(* Logix 5000 project; controller cal1615 1756-L62 rev 20.19; software revision 20.05; part 35 of 81 *)
(* tags used below, declared in another part *)
   FAULT : BOOL;   // Fault AFI
   HMI : BOOL;   // AFI HMI
   p01_param_oven_timer_presets : DINT[32];   // System Parameter Oven Timer Presets
   p01_sys_lc : Limit_Clamp;   // Zone 1 Misc Control Limit Clamp
   p01r09_pb_global_reset : BOOL;   // System Modes PB: Global Fault Reset
   p01r11 : routine;   // System Timer Presets
   p02_real_from_hmi : hmi_real;   // MOP HMI Iface Real from HMI
   p19_dint_to_hmi : DINT[16];
   p19_param_pid1_ff : REAL;
   p19_param_pid1_kd : REAL;
   p19_param_pid1_ki : REAL;
   p19_param_pid1_kp : REAL;
   p19_param_pid2_ff : REAL;
   p19_param_pid2_kd : REAL;
   p19_param_pid2_ki : REAL;
   p19_param_pid2_kp : REAL;
   p19_param_tc01_dev : REAL;
   p19_param_tc01z : REAL;   // Advanced Cooling Parameter Control Temperature 1 Zero Offset
   p19_param_tc02z : REAL;   // Advanced Cooling Parameter Control Temperature 2 Zero Offset
   p19_param_zone_pressure : REAL;   // Advanced Cooling Parameter Minimum Pressusre
   p19r01 : routine;   // Advanced Cooling Main
   p19r02_timer_warning : TIMER[4];   // Advanced Cooling Warning Delay
   p19r07 : routine;   // Advanced Cooling Alarms
   p19r07_timer_fault : TIMER[4];   // Advanced Cooling Alarms Fault Delay
   p19r07_timer_warning : TIMER[4];   // Advanced Cooling Alarms Warning Delay
   p19r08 : routine;   // Advanced Cooling Warnings
   p19r08_timer_fault : TIMER[4];   // Advanced Cooling Warnings Fault Delay
   p19r08_timer_warning : TIMER[4];   // Advanced Cooling Warnings Warning Delay
   p19r09 : routine;   // Advanced Cooling Modes
   p19r09_timer_fault : TIMER[4];   // Advanced Cooling Modes Fault Delay
   p19r09_timer_warning : TIMER[4];   // Advanced Cooling Modes Warning Delay
   p19r10 : routine;   // Advanced Cooling Parameters
   p19r10_timer_fault : TIMER[4];   // Advanced Cooling Parameters Fault Delay
   p19r30 : routine;   // Advanced Cooling Temperature Control
   p19r30_cv_man_sp : REAL;   // Advanced Cooling Manual Control Valve Setpoint
   p19r30_timer_fault : TIMER[4];   // Advanced Cooling Temperature Control Thermocouple Failure
   p19r30_timer_warning : TIMER[4];   // Advanced Cooling Temperature Control Warning Delay
   p19r31 : routine;   // Advanced Cooling Pump
   p19r31_timer_fault : TIMER[4];   // Advanced Cooling Pump Fault Delay
(* P19_Advanced_Cooling, continued *)

ROUTINE R07_Alarms   (* ladder *)
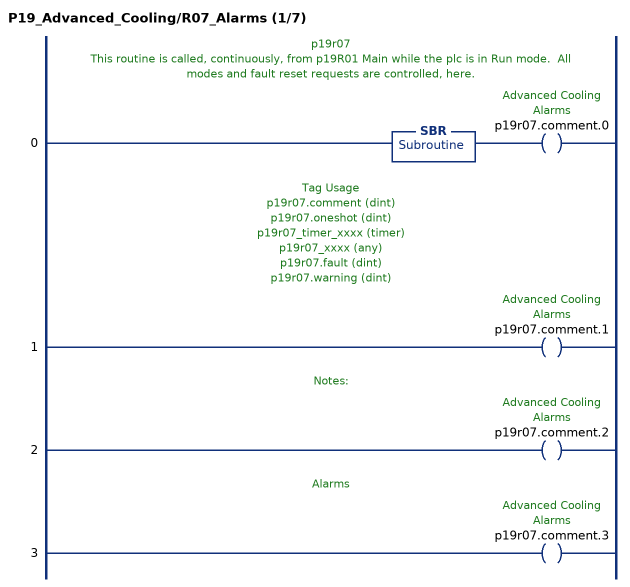
   // p19r07
   // This routine is called, continuously, from p19R01 Main while the plc is in Run mode.  All modes and fault reset requests are controlled, here.
   0: SBR()OTE(p19r07.comment.0);
   // Tag Usage
   // p19r07.comment (dint)
   // p19r07.oneshot (dint)
   // p19r07_timer_xxxx (timer)
   // p19r07_xxxx (any)
   // p19r07.fault (dint)
   // p19r07.warning (dint)
   1: OTE(p19r07.comment.1);
   // Notes:
   2: OTE(p19r07.comment.2);
   // Alarms
   3: OTE(p19r07.comment.3);
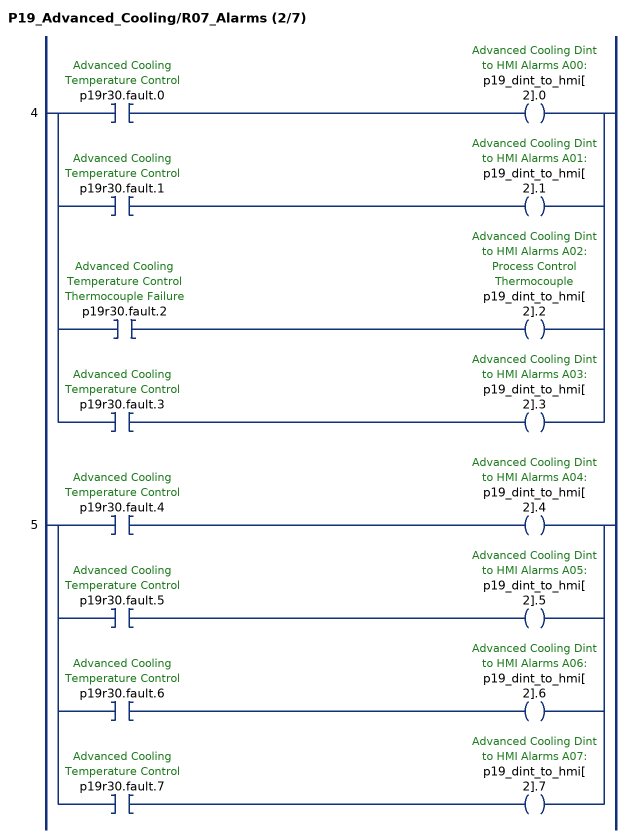
   4: [XIC(p19r30.fault.0) OTE(p19_dint_to_hmi[2].0) ,XIC(p19r30.fault.1) OTE(p19_dint_to_hmi[2].1) ,XIC(p19r30.fault.2) OTE(p19_dint_to_hmi[2].2) ,XIC(p19r30.fault.3) OTE(p19_dint_to_hmi[2].3) ];
   5: [XIC(p19r30.fault.4) OTE(p19_dint_to_hmi[2].4) ,XIC(p19r30.fault.5) OTE(p19_dint_to_hmi[2].5) ,XIC(p19r30.fault.6) OTE(p19_dint_to_hmi[2].6) ,XIC(p19r30.fault.7) OTE(p19_dint_to_hmi[2].7) ];
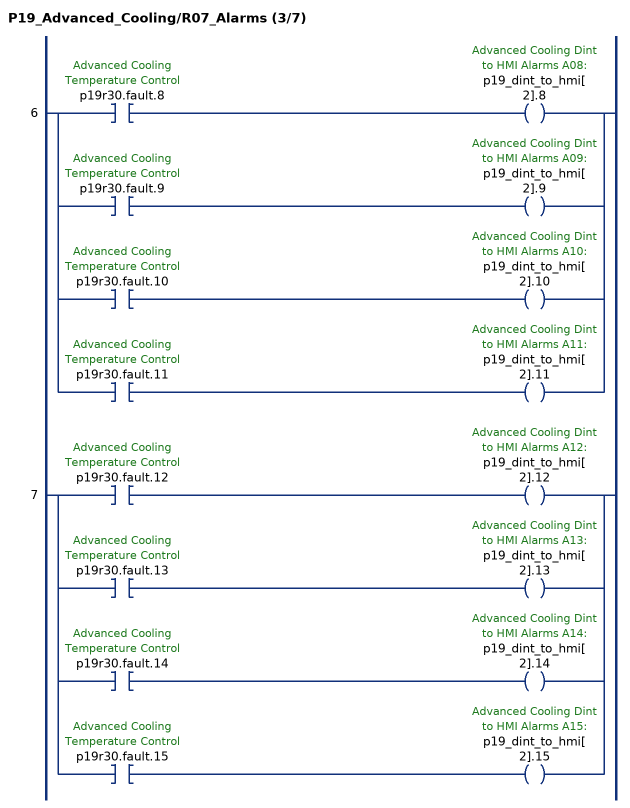
   6: [XIC(p19r30.fault.8) OTE(p19_dint_to_hmi[2].8) ,XIC(p19r30.fault.9) OTE(p19_dint_to_hmi[2].9) ,XIC(p19r30.fault.10) OTE(p19_dint_to_hmi[2].10) ,XIC(p19r30.fault.11) OTE(p19_dint_to_hmi[2].11) ];
   7: [XIC(p19r30.fault.12) OTE(p19_dint_to_hmi[2].12) ,XIC(p19r30.fault.13) OTE(p19_dint_to_hmi[2].13) ,XIC(p19r30.fault.14) OTE(p19_dint_to_hmi[2].14) ,XIC(p19r30.fault.15) OTE(p19_dint_to_hmi[2].15) ];
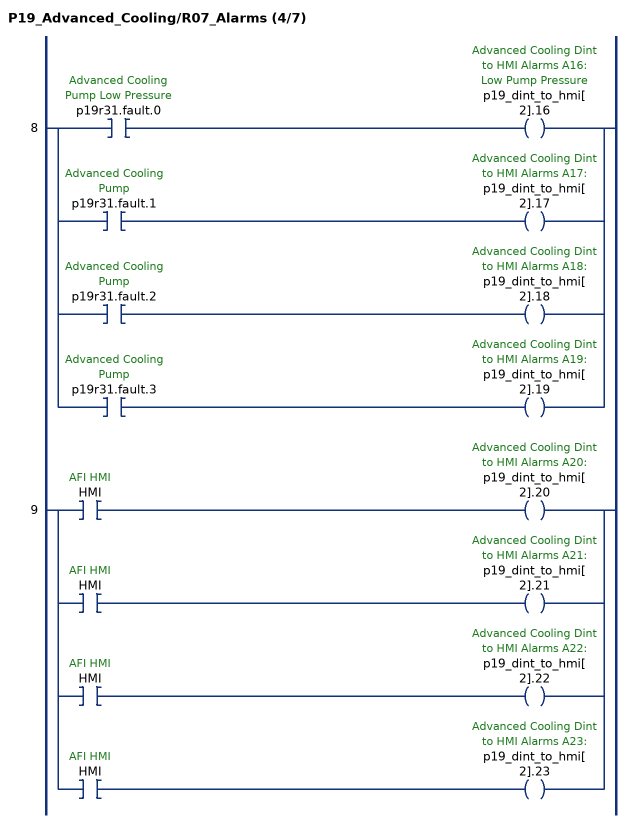
   8: [XIC(p19r31.fault.0) OTE(p19_dint_to_hmi[2].16) ,XIC(p19r31.fault.1) OTE(p19_dint_to_hmi[2].17) ,XIC(p19r31.fault.2) OTE(p19_dint_to_hmi[2].18) ,XIC(p19r31.fault.3) OTE(p19_dint_to_hmi[2].19) ];
   9: [XIC(HMI) OTE(p19_dint_to_hmi[2].20) ,XIC(HMI) OTE(p19_dint_to_hmi[2].21) ,XIC(HMI) OTE(p19_dint_to_hmi[2].22) ,XIC(HMI) OTE(p19_dint_to_hmi[2].23) ];
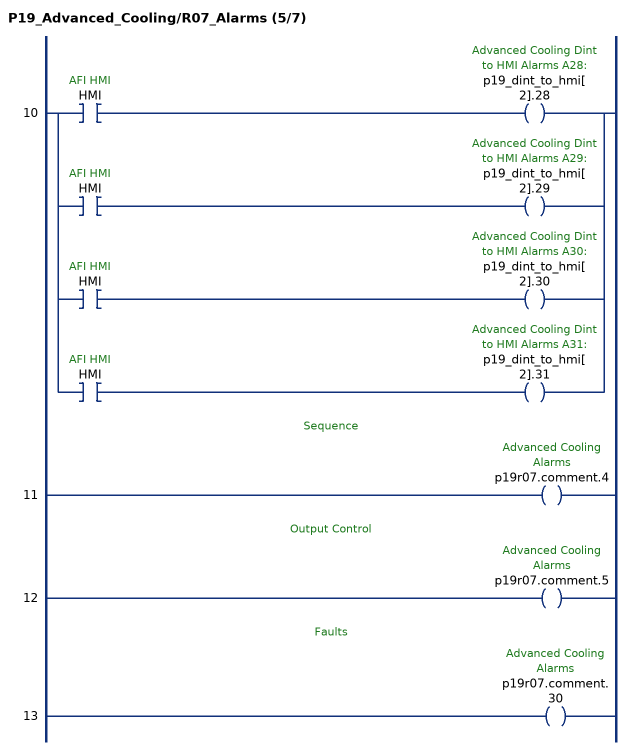
   10: [XIC(HMI) OTE(p19_dint_to_hmi[2].28) ,XIC(HMI) OTE(p19_dint_to_hmi[2].29) ,XIC(HMI) OTE(p19_dint_to_hmi[2].30) ,XIC(HMI) OTE(p19_dint_to_hmi[2].31) ];
   // Sequence
   11: OTE(p19r07.comment.4);
   // Output Control
   12: OTE(p19r07.comment.5);
   // Faults
   13: OTE(p19r07.comment.30);
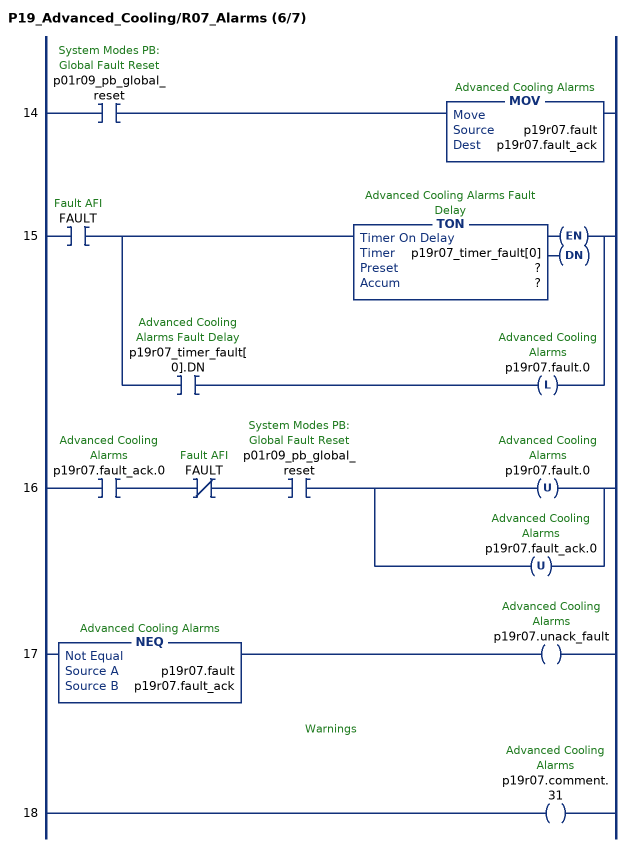
   14: XIC(p01r09_pb_global_reset)MOV(p19r07.fault,p19r07.fault_ack);
   15: XIC(FAULT)[TON(p19r07_timer_fault[0],?,?) ,XIC(p19r07_timer_fault[0].DN) OTL(p19r07.fault.0) ];
   16: XIC(p19r07.fault_ack.0)XIO(FAULT)XIC(p01r09_pb_global_reset)[OTU(p19r07.fault.0) ,OTU(p19r07.fault_ack.0) ];
   17: NEQ(p19r07.fault,p19r07.fault_ack)OTE(p19r07.unack_fault);
   // Warnings
   18: OTE(p19r07.comment.31);
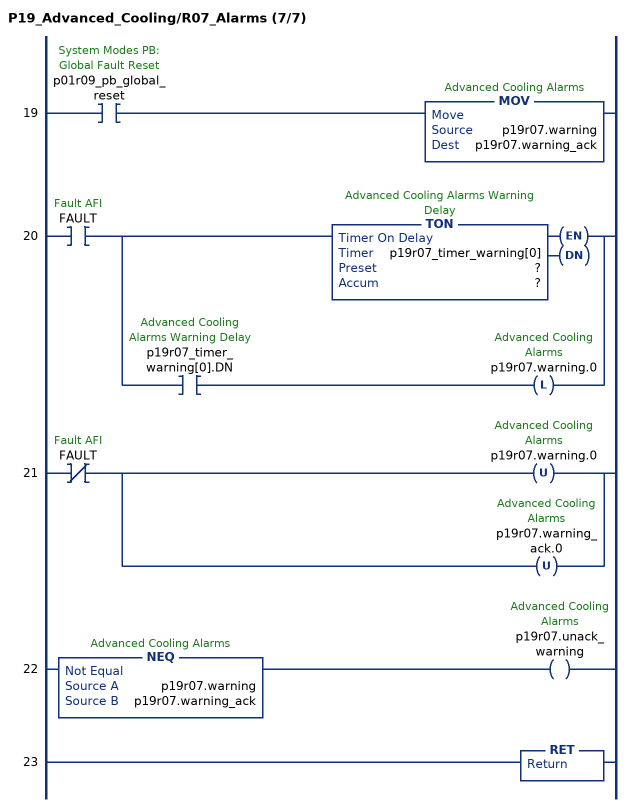
   19: XIC(p01r09_pb_global_reset)MOV(p19r07.warning,p19r07.warning_ack);
   20: XIC(FAULT)[TON(p19r07_timer_warning[0],?,?) ,XIC(p19r07_timer_warning[0].DN) OTL(p19r07.warning.0) ];
   21: XIO(FAULT)[OTU(p19r07.warning.0) ,OTU(p19r07.warning_ack.0) ];
   22: NEQ(p19r07.warning,p19r07.warning_ack)OTE(p19r07.unack_warning);
   23: RET();
END_ROUTINE

ROUTINE R08_Warnings   (* ladder *)
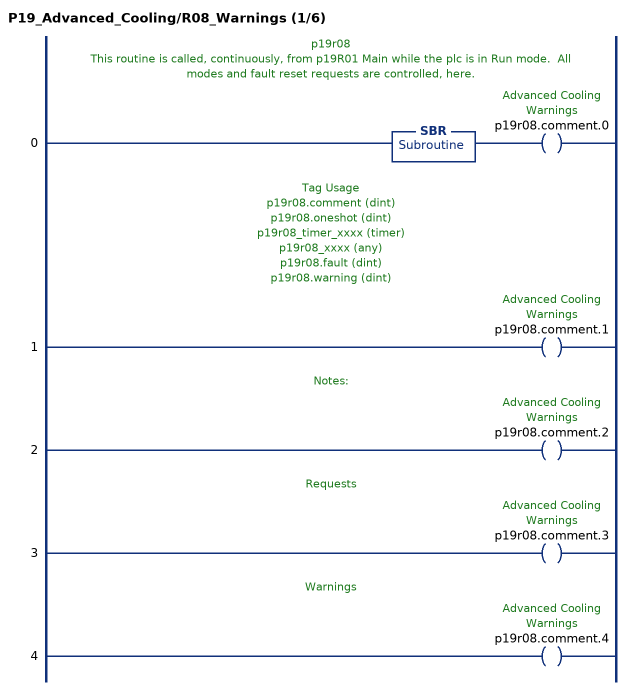
   // p19r08
   // This routine is called, continuously, from p19R01 Main while the plc is in Run mode.  All modes and fault reset requests are controlled, here.
   0: SBR()OTE(p19r08.comment.0);
   // Tag Usage
   // p19r08.comment (dint)
   // p19r08.oneshot (dint)
   // p19r08_timer_xxxx (timer)
   // p19r08_xxxx (any)
   // p19r08.fault (dint)
   // p19r08.warning (dint)
   1: OTE(p19r08.comment.1);
   // Notes:
   2: OTE(p19r08.comment.2);
   // Requests
   3: OTE(p19r08.comment.3);
   // Warnings
   4: OTE(p19r08.comment.4);
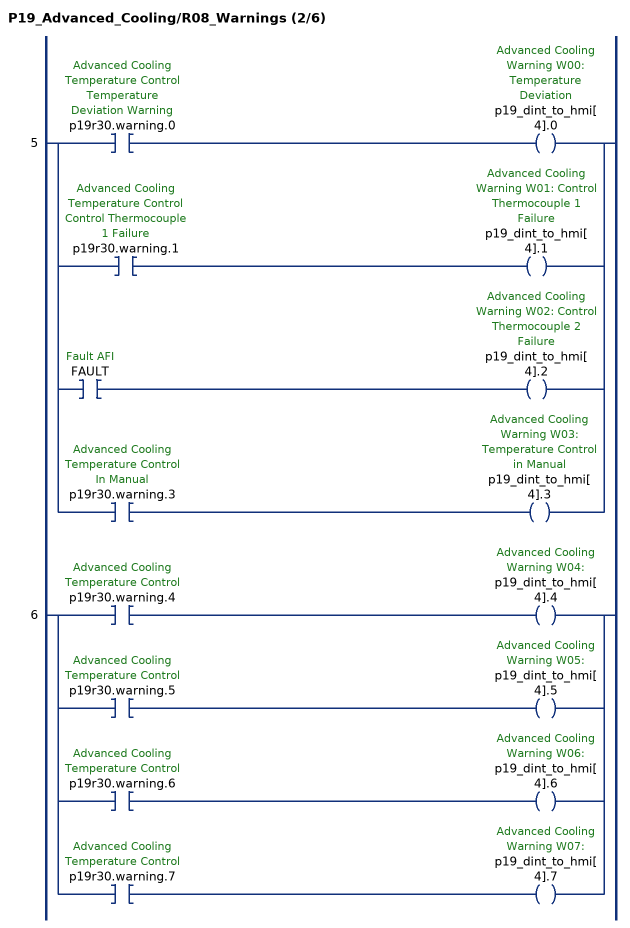
   5: [XIC(p19r30.warning.0) OTE(p19_dint_to_hmi[4].0) ,XIC(p19r30.warning.1) OTE(p19_dint_to_hmi[4].1) ,XIC(FAULT) OTE(p19_dint_to_hmi[4].2) ,XIC(p19r30.warning.3) OTE(p19_dint_to_hmi[4].3) ];
   6: [XIC(p19r30.warning.4) OTE(p19_dint_to_hmi[4].4) ,XIC(p19r30.warning.5) OTE(p19_dint_to_hmi[4].5) ,XIC(p19r30.warning.6) OTE(p19_dint_to_hmi[4].6) ,XIC(p19r30.warning.7) OTE(p19_dint_to_hmi[4].7) ];
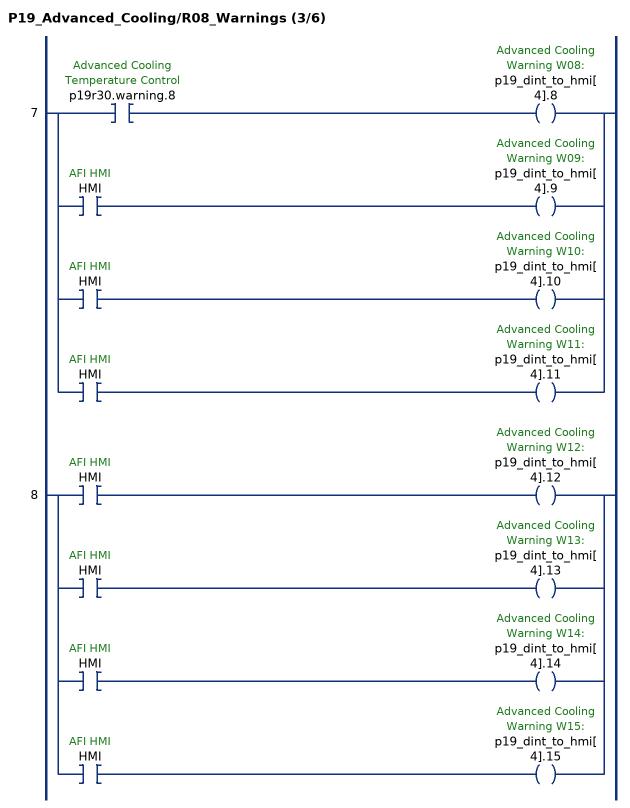
   7: [XIC(p19r30.warning.8) OTE(p19_dint_to_hmi[4].8) ,XIC(HMI) OTE(p19_dint_to_hmi[4].9) ,XIC(HMI) OTE(p19_dint_to_hmi[4].10) ,XIC(HMI) OTE(p19_dint_to_hmi[4].11) ];
   8: [XIC(HMI) OTE(p19_dint_to_hmi[4].12) ,XIC(HMI) OTE(p19_dint_to_hmi[4].13) ,XIC(HMI) OTE(p19_dint_to_hmi[4].14) ,XIC(HMI) OTE(p19_dint_to_hmi[4].15) ];
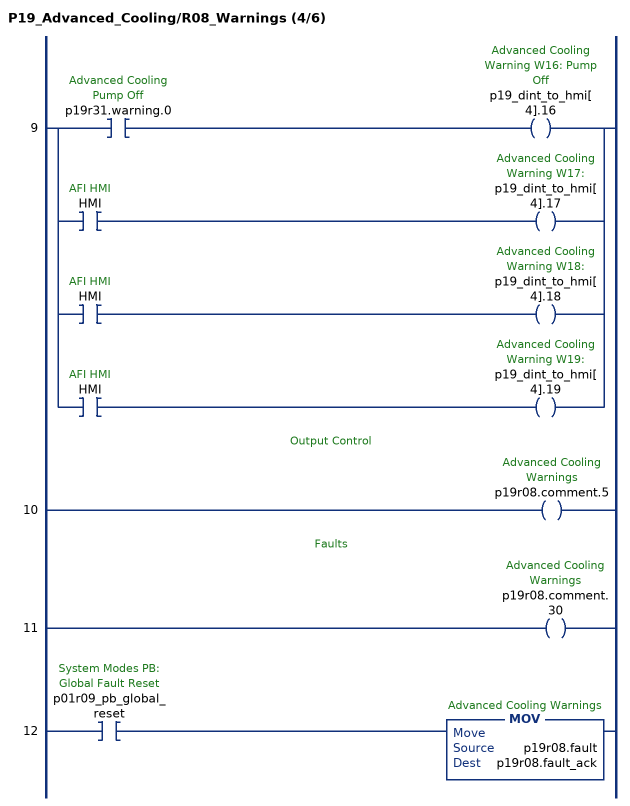
   9: [XIC(p19r31.warning.0) OTE(p19_dint_to_hmi[4].16) ,XIC(HMI) OTE(p19_dint_to_hmi[4].17) ,XIC(HMI) OTE(p19_dint_to_hmi[4].18) ,XIC(HMI) OTE(p19_dint_to_hmi[4].19) ];
   // Output Control
   10: OTE(p19r08.comment.5);
   // Faults
   11: OTE(p19r08.comment.30);
   12: XIC(p01r09_pb_global_reset)MOV(p19r08.fault,p19r08.fault_ack);
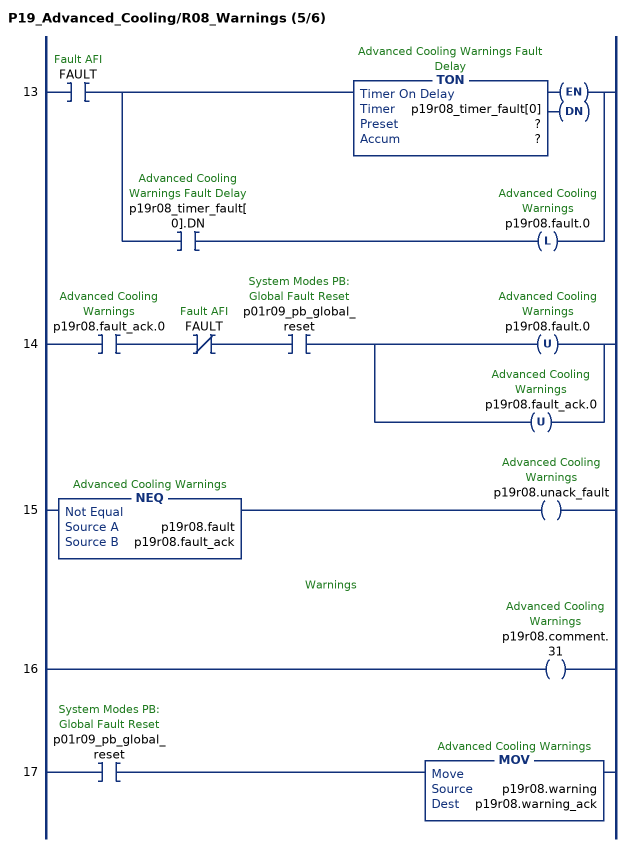
   13: XIC(FAULT)[TON(p19r08_timer_fault[0],?,?) ,XIC(p19r08_timer_fault[0].DN) OTL(p19r08.fault.0) ];
   14: XIC(p19r08.fault_ack.0)XIO(FAULT)XIC(p01r09_pb_global_reset)[OTU(p19r08.fault.0) ,OTU(p19r08.fault_ack.0) ];
   15: NEQ(p19r08.fault,p19r08.fault_ack)OTE(p19r08.unack_fault);
   // Warnings
   16: OTE(p19r08.comment.31);
   17: XIC(p01r09_pb_global_reset)MOV(p19r08.warning,p19r08.warning_ack);
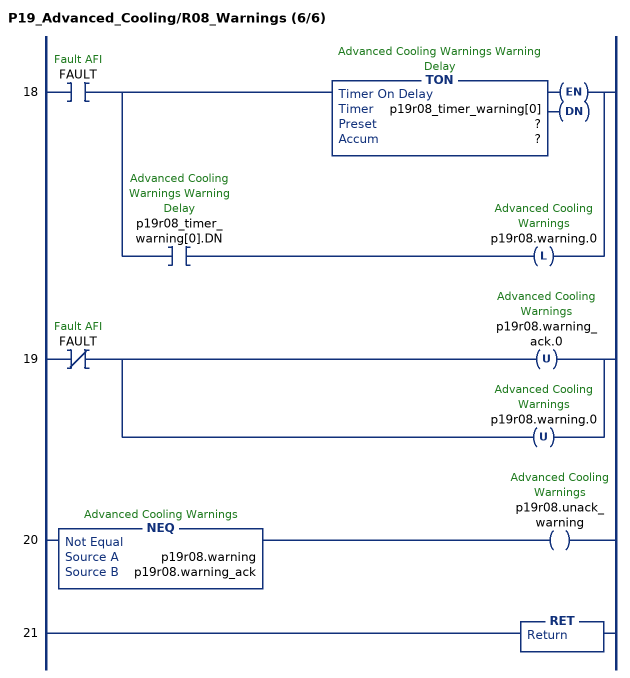
   18: XIC(FAULT)[TON(p19r08_timer_warning[0],?,?) ,XIC(p19r08_timer_warning[0].DN) OTL(p19r08.warning.0) ];
   19: XIO(FAULT)[OTU(p19r08.warning_ack.0) ,OTU(p19r08.warning.0) ];
   20: NEQ(p19r08.warning,p19r08.warning_ack)OTE(p19r08.unack_warning);
   21: RET();
END_ROUTINE

ROUTINE R09_Modes   (* ladder *)
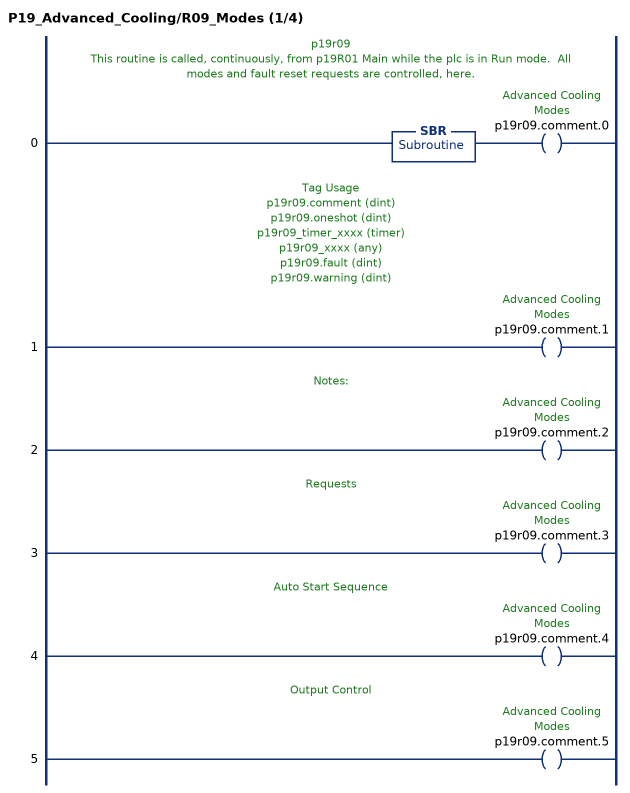
   // p19r09
   // This routine is called, continuously, from p19R01 Main while the plc is in Run mode.  All modes and fault reset requests are controlled, here.
   0: SBR()OTE(p19r09.comment.0);
   // Tag Usage
   // p19r09.comment (dint)
   // p19r09.oneshot (dint)
   // p19r09_timer_xxxx (timer)
   // p19r09_xxxx (any)
   // p19r09.fault (dint)
   // p19r09.warning (dint)
   1: OTE(p19r09.comment.1);
   // Notes:
   2: OTE(p19r09.comment.2);
   // Requests
   3: OTE(p19r09.comment.3);
   // Auto Start Sequence
   4: OTE(p19r09.comment.4);
   // Output Control
   5: OTE(p19r09.comment.5);
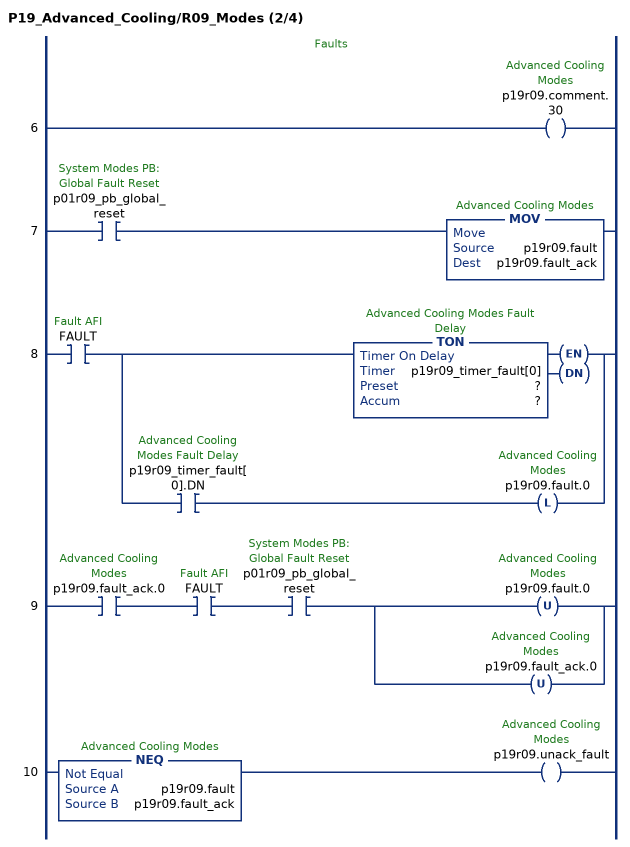
   // Faults
   6: OTE(p19r09.comment.30);
   7: XIC(p01r09_pb_global_reset)MOV(p19r09.fault,p19r09.fault_ack);
   8: XIC(FAULT)[TON(p19r09_timer_fault[0],?,?) ,XIC(p19r09_timer_fault[0].DN) OTL(p19r09.fault.0) ];
   9: XIC(p19r09.fault_ack.0)XIC(FAULT)XIC(p01r09_pb_global_reset)[OTU(p19r09.fault.0) ,OTU(p19r09.fault_ack.0) ];
   10: NEQ(p19r09.fault,p19r09.fault_ack)OTE(p19r09.unack_fault);
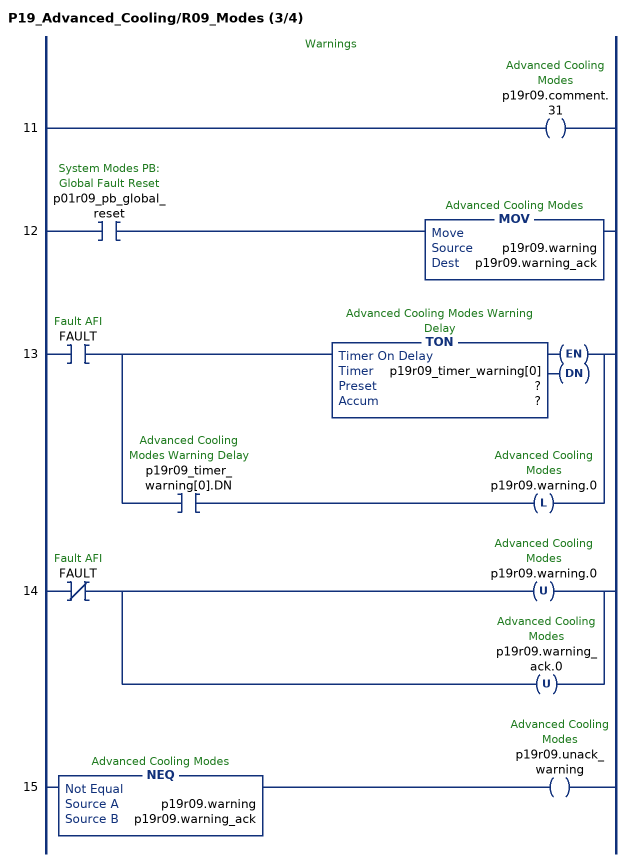
   // Warnings
   11: OTE(p19r09.comment.31);
   12: XIC(p01r09_pb_global_reset)MOV(p19r09.warning,p19r09.warning_ack);
   13: XIC(FAULT)[TON(p19r09_timer_warning[0],?,?) ,XIC(p19r09_timer_warning[0].DN) OTL(p19r09.warning.0) ];
   14: XIO(FAULT)[OTU(p19r09.warning.0) ,OTU(p19r09.warning_ack.0) ];
   15: NEQ(p19r09.warning,p19r09.warning_ack)OTE(p19r09.unack_warning);
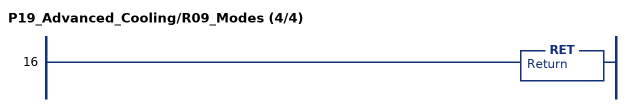
   16: RET();
END_ROUTINE

ROUTINE R10_Parameters   (* ladder *)
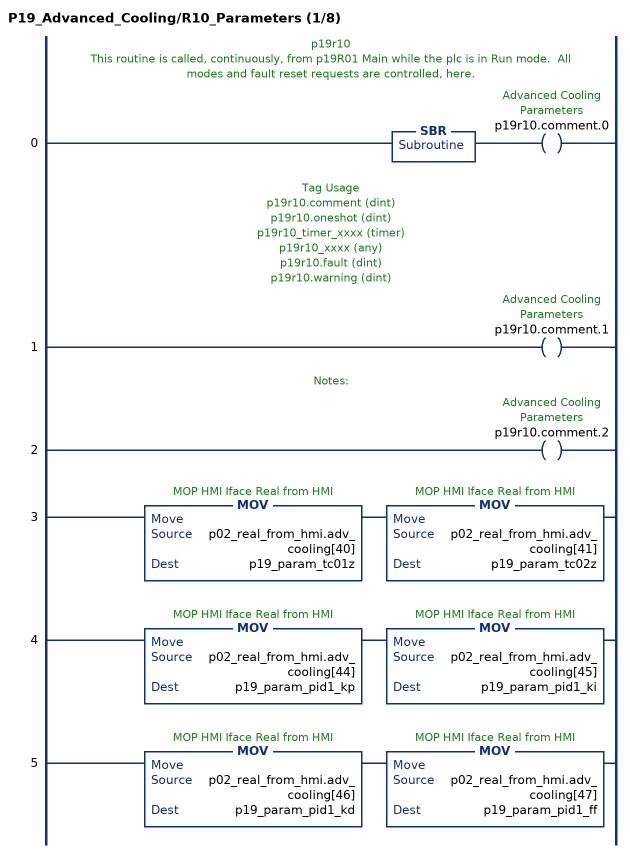
   // p19r10
   // This routine is called, continuously, from p19R01 Main while the plc is in Run mode.  All modes and fault reset requests are controlled, here.
   0: SBR()OTE(p19r10.comment.0);
   // Tag Usage
   // p19r10.comment (dint)
   // p19r10.oneshot (dint)
   // p19r10_timer_xxxx (timer)
   // p19r10_xxxx (any)
   // p19r10.fault (dint)
   // p19r10.warning (dint)
   1: OTE(p19r10.comment.1);
   // Notes:
   2: OTE(p19r10.comment.2);
   3: MOV(p02_real_from_hmi.adv_cooling[40],p19_param_tc01z)MOV(p02_real_from_hmi.adv_cooling[41],p19_param_tc02z);
   4: MOV(p02_real_from_hmi.adv_cooling[44],p19_param_pid1_kp)MOV(p02_real_from_hmi.adv_cooling[45],p19_param_pid1_ki);
   5: MOV(p02_real_from_hmi.adv_cooling[46],p19_param_pid1_kd)MOV(p02_real_from_hmi.adv_cooling[47],p19_param_pid1_ff);
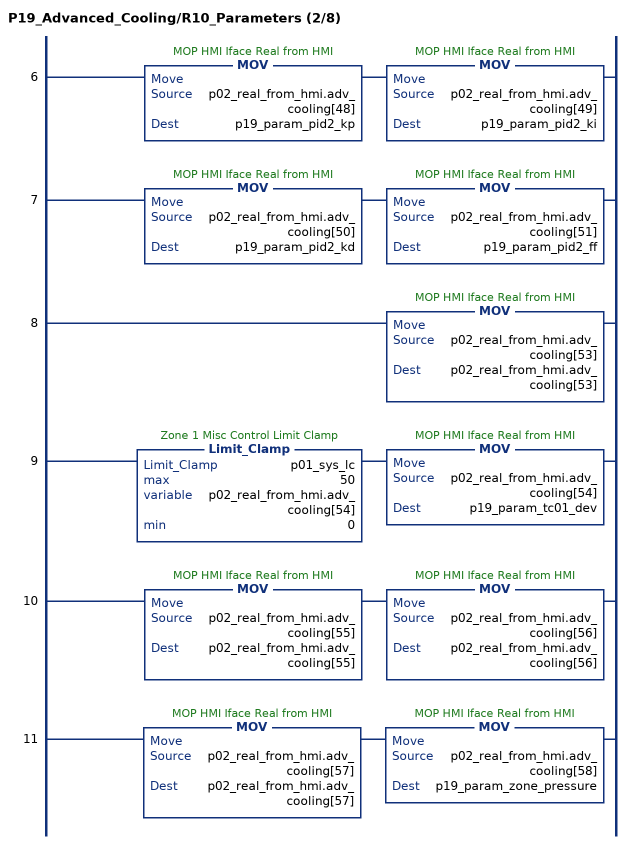
   6: MOV(p02_real_from_hmi.adv_cooling[48],p19_param_pid2_kp)MOV(p02_real_from_hmi.adv_cooling[49],p19_param_pid2_ki);
   7: MOV(p02_real_from_hmi.adv_cooling[50],p19_param_pid2_kd)MOV(p02_real_from_hmi.adv_cooling[51],p19_param_pid2_ff);
   8: MOV(p02_real_from_hmi.adv_cooling[53],p02_real_from_hmi.adv_cooling[53]);
   9: Limit_Clamp(p01_sys_lc,50,p02_real_from_hmi.adv_cooling[54],0)MOV(p02_real_from_hmi.adv_cooling[54],p19_param_tc01_dev);
   10: MOV(p02_real_from_hmi.adv_cooling[55],p02_real_from_hmi.adv_cooling[55])MOV(p02_real_from_hmi.adv_cooling[56],p02_real_from_hmi.adv_cooling[56]);
   11: MOV(p02_real_from_hmi.adv_cooling[57],p02_real_from_hmi.adv_cooling[57])MOV(p02_real_from_hmi.adv_cooling[58],p19_param_zone_pressure);
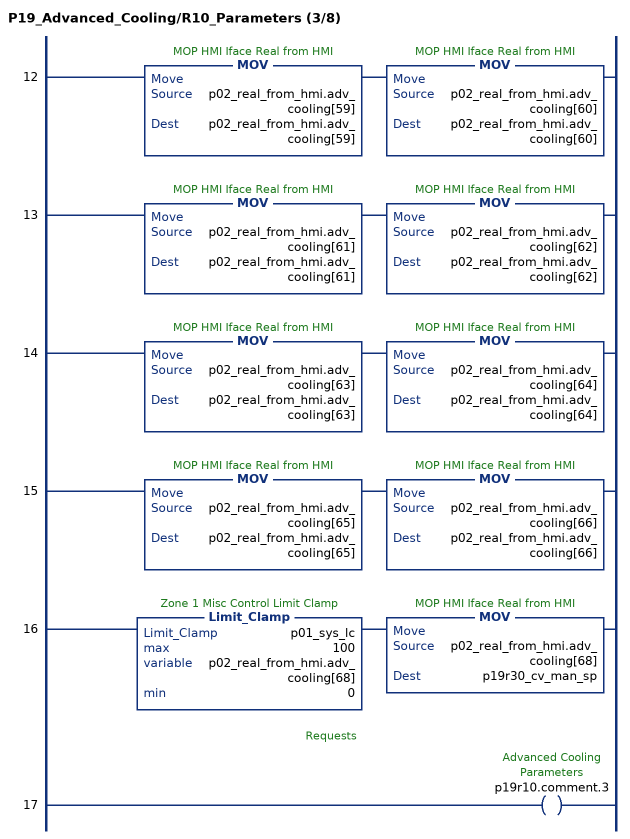
   12: MOV(p02_real_from_hmi.adv_cooling[59],p02_real_from_hmi.adv_cooling[59])MOV(p02_real_from_hmi.adv_cooling[60],p02_real_from_hmi.adv_cooling[60]);
   13: MOV(p02_real_from_hmi.adv_cooling[61],p02_real_from_hmi.adv_cooling[61])MOV(p02_real_from_hmi.adv_cooling[62],p02_real_from_hmi.adv_cooling[62]);
   14: MOV(p02_real_from_hmi.adv_cooling[63],p02_real_from_hmi.adv_cooling[63])MOV(p02_real_from_hmi.adv_cooling[64],p02_real_from_hmi.adv_cooling[64]);
   15: MOV(p02_real_from_hmi.adv_cooling[65],p02_real_from_hmi.adv_cooling[65])MOV(p02_real_from_hmi.adv_cooling[66],p02_real_from_hmi.adv_cooling[66]);
   16: Limit_Clamp(p01_sys_lc,100,p02_real_from_hmi.adv_cooling[68],0)MOV(p02_real_from_hmi.adv_cooling[68],p19r30_cv_man_sp);
   // Requests
   17: OTE(p19r10.comment.3);
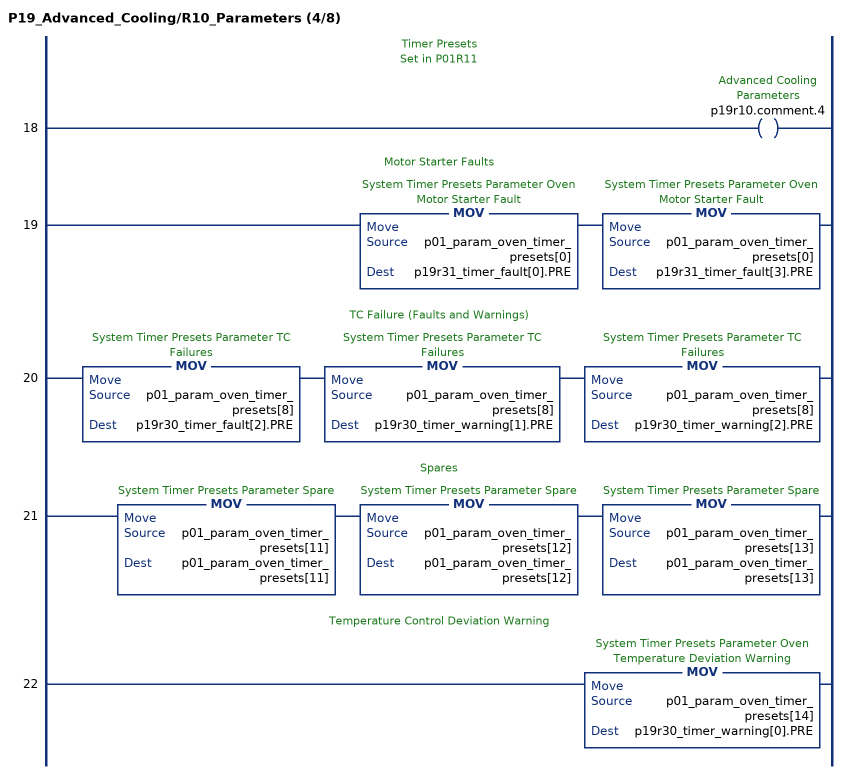
   // Timer Presets
   // Set in P01R11
   18: OTE(p19r10.comment.4);
   // Motor Starter Faults
   19: MOV(p01_param_oven_timer_presets[0],p19r31_timer_fault[0].PRE)MOV(p01_param_oven_timer_presets[0],p19r31_timer_fault[3].PRE);
   // TC Failure (Faults and Warnings)
   20: MOV(p01_param_oven_timer_presets[8],p19r30_timer_fault[2].PRE)MOV(p01_param_oven_timer_presets[8],p19r30_timer_warning[1].PRE)MOV(p01_param_oven_timer_presets[8],p19r30_timer_warning[2].PRE);
   // Spares
   21: MOV(p01_param_oven_timer_presets[11],p01_param_oven_timer_presets[11])MOV(p01_param_oven_timer_presets[12],p01_param_oven_timer_presets[12])MOV(p01_param_oven_timer_presets[13],p01_param_oven_timer_presets[13]);
   // Temperature Control Deviation Warning
   22: MOV(p01_param_oven_timer_presets[14],p19r30_timer_warning[0].PRE);
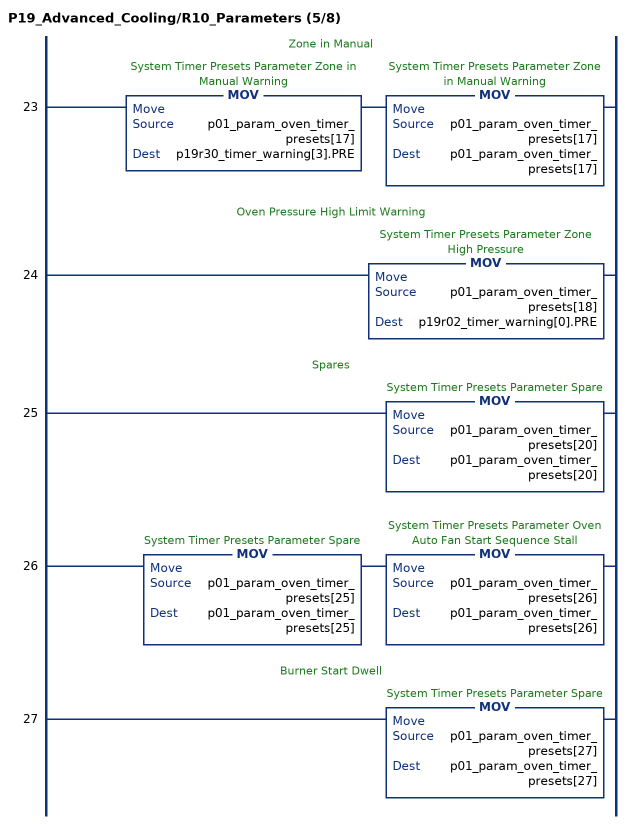
   // Zone in Manual
   23: MOV(p01_param_oven_timer_presets[17],p19r30_timer_warning[3].PRE)MOV(p01_param_oven_timer_presets[17],p01_param_oven_timer_presets[17]);
   // Oven Pressure High Limit Warning
   24: MOV(p01_param_oven_timer_presets[18],p19r02_timer_warning[0].PRE);
   // Spares
   25: MOV(p01_param_oven_timer_presets[20],p01_param_oven_timer_presets[20]);
   26: MOV(p01_param_oven_timer_presets[25],p01_param_oven_timer_presets[25])MOV(p01_param_oven_timer_presets[26],p01_param_oven_timer_presets[26]);
   // Burner Start Dwell
   27: MOV(p01_param_oven_timer_presets[27],p01_param_oven_timer_presets[27]);
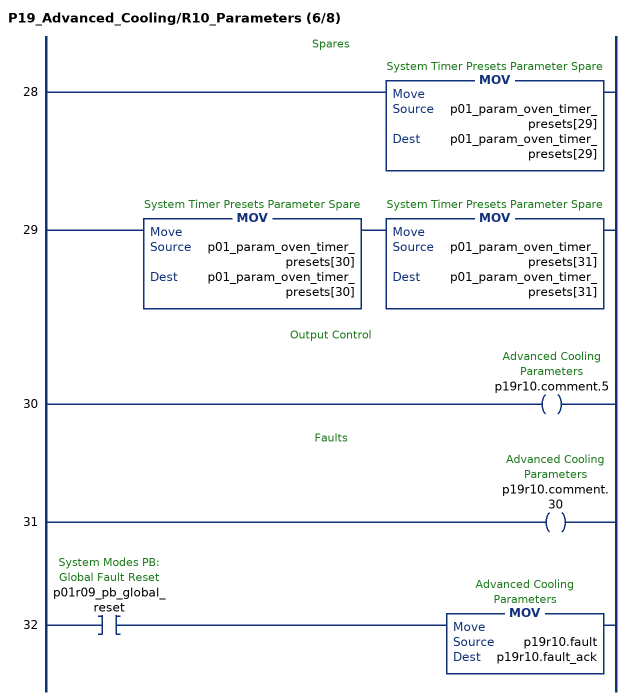
   // Spares
   28: MOV(p01_param_oven_timer_presets[29],p01_param_oven_timer_presets[29]);
   29: MOV(p01_param_oven_timer_presets[30],p01_param_oven_timer_presets[30])MOV(p01_param_oven_timer_presets[31],p01_param_oven_timer_presets[31]);
   // Output Control
   30: OTE(p19r10.comment.5);
   // Faults
   31: OTE(p19r10.comment.30);
   32: XIC(p01r09_pb_global_reset)MOV(p19r10.fault,p19r10.fault_ack);
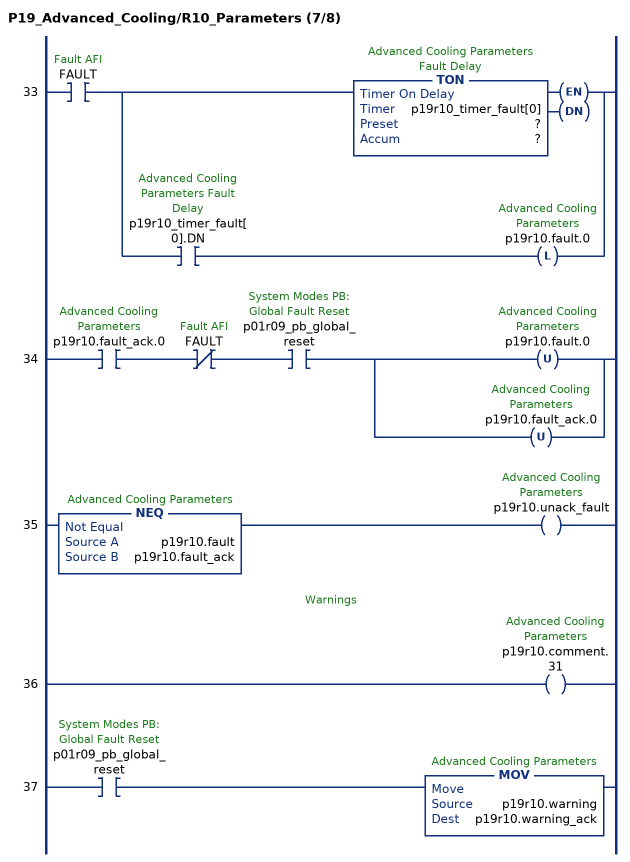
   33: XIC(FAULT)[TON(p19r10_timer_fault[0],?,?) ,XIC(p19r10_timer_fault[0].DN) OTL(p19r10.fault.0) ];
   34: XIC(p19r10.fault_ack.0)XIO(FAULT)XIC(p01r09_pb_global_reset)[OTU(p19r10.fault.0) ,OTU(p19r10.fault_ack.0) ];
   35: NEQ(p19r10.fault,p19r10.fault_ack)OTE(p19r10.unack_fault);
   // Warnings
   36: OTE(p19r10.comment.31);
   37: XIC(p01r09_pb_global_reset)MOV(p19r10.warning,p19r10.warning_ack);
